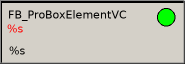
VISUALIZATION V_Element_Base  // 185x64
VAR_IN_OUT
	{attribute 'VAR_IN_OUT_AS_POINTER'}
	fbFunction		: FB_ProBoxElementBase;	
END_VAR
    Rectangle (0,1 185x63), colour toggle: fbFunction.fbProBoxMotorControl_12.Run
    Rectangle (6,41 143x20), "%s", text variable: fbFunction.ConfigElement.ElementName
    Label (5,5 158x20), "FB_ProBoxElementVC"
    Rectangle (4,19 161x20), "%s", tooltip "%s", text variable: fbFunction.ElementData.ErrorData.Error.ErrorCode.Conv, invisible if: fbFunction.ElementData.ErrorData.Error.ErrorCode.Conv = 0
        p4168582468: fbFunction.ElementData.ErrorData.Error.ErrorParam
    Ellipse (157,8 18x18), colour toggle: NOT fbFunction.HW_Inputs.MotorUnitOK
END_VISUALIZATION

(* stored: Version 1.1.0.1, ProductVersion 3.1.4024.9
   Visu V_Element_Base: Id {32c1623f-12e4-469f-b417-d5fea3d9e8d9} *)
